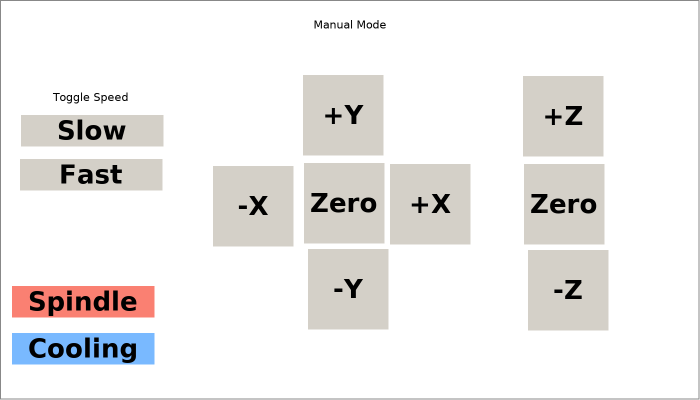
VISUALIZATION V_ManualMode  // 700x400
VAR_IN_OUT
	HMI : ST_PackMLBaseModule_HMI;
END_VAR
    RoundedRectangle (304,163 80x80), "Zero"
        OnMouseClick: execute { HMI.Command.State := E_PMLCommand.ePMLCommand_Clear; }
    Label (0,0 700x50), "Manual Mode"
    RoundedRectangle (213,166 80x80), "-X"
        OnMouseClick: execute { HMI.Command.State := E_PMLCommand.ePMLCommand_Clear; }
    RoundedRectangle (390,164 80x80), "+X"
        OnMouseClick: execute { HMI.Command.State := E_PMLCommand.ePMLCommand_Clear; }
    RoundedRectangle (303,75 80x80), "+Y"
        OnMouseClick: execute { HMI.Command.State := E_PMLCommand.ePMLCommand_Clear; }
    RoundedRectangle (308,249 80x80), "-Y"
        OnMouseClick: execute { HMI.Command.State := E_PMLCommand.ePMLCommand_Clear; }
    RoundedRectangle (524,164 80x80), "Zero"
        OnMouseClick: execute { HMI.Command.State := E_PMLCommand.ePMLCommand_Clear; }
    RoundedRectangle (523,76 80x80), "+Z"
        OnMouseClick: execute { HMI.Command.State := E_PMLCommand.ePMLCommand_Clear; }
    RoundedRectangle (528,250 80x80), "-Z"
        OnMouseClick: execute { HMI.Command.State := E_PMLCommand.ePMLCommand_Clear; }
    Label (16,66 150x63), "Toggle Speed"
    RoundedRectangle (21,115 142x31), "Slow"
        OnMouseClick: execute { HMI.Command.State := E_PMLCommand.ePMLCommand_Clear; }
    RoundedRectangle (20,159 142x31), "Fast"
        OnMouseClick: execute { HMI.Command.State := E_PMLCommand.ePMLCommand_Clear; }
    RoundedRectangle (12,286 142x31), "Spindle"
        OnMouseClick: execute { HMI.Command.State := E_PMLCommand.ePMLCommand_Clear; }
    RoundedRectangle (12,333 142x31), "Cooling"
        OnMouseClick: execute { HMI.Command.State := E_PMLCommand.ePMLCommand_Clear; }
END_VISUALIZATION

(* stored: Version 1.1.0.1, ProductVersion 3.1.4024.15
   Visu V_ManualMode: Id {5eb24302-7c74-4cb0-913c-af4cad05dac4} *)
